Yaskawa INFORM job: R1_W18,19,21(0,0)_KM-OKNEW.JBI

/JOB
//NAME R1_W18,19,21(0,0)_KM-OKNEW
///FOLDERNAME KRIS-SCIANA
//POS
///NPOS 59,59,0,3,0,0
///TOOL 0
///POSTYPE PULSE
///PULSE
C00000=-165945,-65747,-78398,-11730,94813,86069
C00001=-225738,-29129,-36820,-61092,45172,49948
C00002=-227041,-26413,-34946,-60254,44485,49501
C00003=-227207,-24592,-33670,-60039,44458,49378
C00004=-237533,-37402,-42560,-38701,28295,39081
C00005=-229553,-27860,-24718,-81378,37631,57193
C00006=-236638,-41709,-45274,-40385,28277,39894
C00007=-227197,-30656,-28257,-80893,39459,56892
C00008=-224091,-34376,-30000,-82400,41545,57754
C00009=-209639,-77270,-46477,-91612,78281,60493
C00010=178105,-72497,-44360,72515,40978,-24705
C00011=157900,67762,47803,76590,91490,-60139
C00012=160086,65038,44626,76467,90101,-59697
C00013=160971,64038,43468,76405,89533,-59530
C00014=161808,65957,45694,76334,88844,-59627
C00015=160971,64038,43468,76405,89533,-59530
C00016=160746,61033,49335,86208,88631,-60628
C00017=161214,57780,45635,86203,88352,-60332
C00018=160746,61033,49335,86208,88631,-60628
C00019=159860,62185,50950,86211,89235,-60844
C00020=157670,65355,55356,86172,90720,-61418
C00021=161021,60847,32788,71661,91289,-58028
C00022=158071,42272,26850,85179,79726,-64183
C00023=159982,40910,25376,84977,78370,-64008
C00024=160407,59632,31901,71739,91677,-58132
C00025=160676,63082,35844,71667,91272,-58387
C00026=160022,52515,61592,88250,76818,-71686
C00027=151897,58426,66630,87129,82620,-71919
C00028=158751,51722,59033,87847,77807,-71164
C00029=159892,50938,58162,87958,76997,-71072
C00030=160407,59632,31901,71739,91677,-58132
C00031=160676,63082,35844,71667,91272,-58387
C00032=160063,48160,52262,87506,77036,-70029
C00033=151932,45808,25021,85459,84488,-63059
C00034=157434,41112,20051,84712,80618,-62540
C00035=160036,40278,19462,84376,78747,-62460
C00036=160407,59632,31901,71739,91677,-58132
C00037=160676,63082,35844,71667,91272,-58387
C00038=160053,50810,58014,87970,76885,-71060
C00039=156942,58566,66790,87841,79014,-71800
C00040=148876,27456,33542,86429,85194,-69951
C00041=224712,-65391,-70566,-27443,33176,35029
C00042=213770,-36542,-34460,77474,7084,-9175
C00043=213911,-28559,-27626,78111,6960,-9462
C00044=226738,-22872,-44138,-26151,38823,34122
C00045=225474,-24610,-45368,-24938,38325,33575
C00046=213819,-17629,4736,154767,14347,-43948
C00047=214272,-23134,1814,157793,15117,-45305
C00048=214272,-33613,-26176,108147,6753,-22913
C00049=214465,-33157,-25875,108062,6602,-22875
C00050=214484,-33168,-25884,108106,6590,-22894
C00051=214462,-14862,18245,165247,20516,-48770
C00052=217554,-35080,-3939,169426,16769,-50400
C00053=215729,-48765,-65733,21008,15669,16203
C00054=214456,-35235,-57699,21691,17865,16014
C00055=214365,-32785,-25079,110368,6760,-23908
C00056=218232,-57197,-39676,150711,6696,-41886
C00057=106022,-135537,-66235,115408,55550,-32403
C00058=10106,-66575,-39760,6607,87446,-74437
BC00000=342908,239,1075157
BC00001=398174,15,1075175
BC00002=398174,15,1075175
BC00003=398174,15,1075175
BC00004=398174,15,1075175
BC00005=398174,15,1075175
BC00006=398174,15,1075175
BC00007=398174,15,1075175
BC00008=398174,15,1075175
BC00009=394883,45674,1071776
BC00010=394883,231390,1071776
BC00011=365912,447627,1041849
BC00012=365912,447627,1041849
BC00013=365912,447627,1041849
BC00014=365912,447627,1041849
BC00015=365912,447627,1041849
BC00016=365912,447627,1041849
BC00017=365912,447627,1041849
BC00018=365912,447627,1041849
BC00019=365912,447627,1041849
BC00020=365912,447627,1041849
BC00021=368384,441548,1075175
BC00022=360608,449199,1075175
BC00023=360608,449199,1075175
BC00024=360608,449199,1075175
BC00025=360608,449199,1075175
BC00026=360608,449199,1075175
BC00027=360608,449199,871920
BC00028=360608,449199,871920
BC00029=360608,449199,871920
BC00030=360608,449199,1075175
BC00031=360608,449199,1075175
BC00032=360608,449199,655426
BC00033=360609,449199,890554
BC00034=360609,449199,890554
BC00035=360608,449199,890556
BC00036=360608,449199,1075175
BC00037=360608,449199,1075175
BC00038=360608,449199,871921
BC00039=360608,449199,871921
BC00040=360608,408502,871921
BC00041=398174,68400,1075175
BC00042=398174,60897,1075175
BC00043=398174,60897,1075175
BC00044=398174,60897,1075175
BC00045=398174,60897,1075175
BC00046=398174,60897,1075175
BC00047=398174,60897,1075175
BC00048=398174,60897,775711
BC00049=392644,57641,759002
BC00050=392644,57641,759002
BC00051=392644,57641,759002
BC00052=392644,57641,759002
BC00053=392644,57641,759002
BC00054=392644,57641,759002
BC00055=392644,57641,759002
BC00056=392644,57641,759002
BC00057=392644,373033,759002
BC00058=221411,449199,1015609
///POSTYPE BASE
///RECTAN
///RCONF 0,0,0,0,1,0,0,0,0,0,0,0,0,0,0,0,0,0,0,0,0,0,0,0
P00006=2.006,1.622,-0.565,0.0000,0.0000,0.0000
///RCONF 0,0,0,0,0,0,0,0,0,0,0,0,0,0,0,0,0,0,0,0,0,0,0,0
P00026=2.644,0.055,-2.583,0.0000,0.0000,0.0000
P00027=2.278,0.099,-4.210,0.0000,0.0000,0.0000
//INST
///DATE 2024/01/25 10:39
///ATTR SC,RW
///GROUP1 RB1,BS1
NOP
SFTOF
MOVJ C00000 BC00000 VJ=100.00
MOVL C00001 BC00001 V=166.7
MOVL C00002 BC00002 V=60.0
REFP 3 C00003 BC00003
CALL JOB:SEARCH-R1
SET P027 P006
SFTON P026
MOVL C00004 BC00004 V=60.0
REFP 3 C00005 BC00005
CALL JOB:SEARCH-R1
SET P027 P006
SFTON P026
MOVL C00006 BC00006 V=60.0
MOVL C00007 BC00007 V=166.7
MOVL C00008 BC00008 V=166.7
SFTOF
MOVJ C00009 BC00009 VJ=40.00
MOVJ C00010 BC00010 VJ=60.00
MOVL C00011 BC00011 V=333.3
MOVL C00012 BC00012 V=166.7
MOVL C00013 BC00013 V=60.0
REFP 3 C00014 BC00014
CALL JOB:SEARCH-R1
SET P026 P006
SFTON P026
MOVL C00015 BC00015 V=60.0
MOVL C00016 BC00016 V=60.0
REFP 3 C00017 BC00017
CALL JOB:SEARCH-R1
SET P026 P006
SFTON P026
MOVL C00018 BC00018 V=60.0
MOVL C00019 BC00019 V=100.0
MOVL C00020 BC00020 V=166.7
'Path S879 (for W18)
SFTOF
SFTOF
SFTON P026
MOVL C00021 BC00021 V=333.3
MOVL C00022 BC00022 V=250.0
MOVL C00023 BC00023 V=166.7 PL=0
REFP 1 C00024 BC00024
REFP 2 C00025 BC00025
MACRO1 MJ#(0) ARGF6
ARCON
MOVL C00026 BC00026 V=13.3
ARCOF
'Path W883_C
SFTOF
SFTON P026
MOVL C00027 BC00027 V=100.0
MOVL C00028 BC00028 V=100.0
MOVL C00029 BC00029 V=100.0 PL=0
REFP 1 C00030 BC00030
REFP 2 C00031 BC00031
MACRO1 MJ#(0) ARGF6
ARCON
MOVL C00032 BC00032 V=13.3
ARCOF
'Path W883_B
SFTOF
SFTON P026
MOVL C00033 BC00033 V=100.0
MOVL C00034 BC00034 V=100.0
MOVL C00035 BC00035 V=100.0 PL=0
REFP 1 C00036 BC00036
REFP 2 C00037 BC00037
MACRO1 MJ#(0) ARGF6
ARCON
MOVL C00038 BC00038 V=13.3
ARCOF
MOVL C00039 BC00039 V=100.0
SFTOF
MOVL C00040 BC00040 V=100.0
MOVL C00041 BC00041 V=333.3
MOVL C00042 BC00042 V=166.7
SFTON P027
MOVL C00043 BC00043 V=100.0 PL=0
REFP 1 C00044 BC00044
REFP 2 C00045 BC00045
MACRO1 MJ#(0) ARGF6
ARCON
MOVL C00046 BC00046 V=12.5
ARCOF
MOVL C00047 BC00047 V=166.7
SFTOF
MOVJ C00048 BC00048 VJ=100.00
SFTON P027
MOVJ C00049 BC00049 VJ=100.00
MACRO1 MJ#(0) ARGF6
MOVL C00050 BC00050 V=50.0 PL=0
ARCON
MOVL C00051 BC00051 V=12.5
ARCOF
TIMER T=1.00
SFTOF
MOVJ C00052 BC00052 VJ=100.00
MOVJ C00053 BC00053 VJ=25.00
SFTON P027
MOVJ C00054 BC00054 VJ=100.00
ARCON
MOVL C00055 BC00055 V=12.5
ARCOF
TIMER T=1.00
SFTOF
MOVL C00056 BC00056 V=166.7
SFTOF
MOVJ C00057 BC00057 VJ=100.00
MOVJ C00058 BC00058 VJ=100.00
END
